(* IEC 61131-3 sources: RL_MAR/experiments/comparison/llm4plc/results/gpt-4o_20260507_114630/20260507_114958, 1 file *)

(* ---- generated_code_iteration_0.st ---- *)
plaintext
START_ST

FUNCTION_BLOCK ShellSortFB
VAR_INPUT
    arr: ARRAY[1..1000] OF DINT; // Input array to be sorted
    sortDirection: BOOL; // Sorting direction (FALSE = ascending, TRUE = descending)
END_VAR

VAR_OUTPUT
    error: BOOL; // Error status (TRUE if an error occurred)
    status: WORD; // Status code
    sorted_arr: ARRAY[1..1000] OF DINT; // Sorted output array
END_VAR

VAR
    state: INT := 0; // Current state of the function block
    N: INT := 1000; // Fixed array size (constant for validation)
    gap: INT; // Gap value for Shell Sort
    i, j: INT; // Loop counters for sorting
    temp: DINT; // Temporary variable for swapping during sorting
END_VAR

// Function block logic
CASE state OF

    // STATE 0: INITIALIZE
    0:
        // Copy input array to output array
        FOR i := 1 TO N DO
            sorted_arr[i] := arr[i];
        END_FOR

        // Validate array size
        IF N <= 1 THEN
            error := TRUE;
            status := 16#8200; // Array size <= 1
            state := 2; // Transition to COMPLETION state
        ELSIF N > 1000 THEN
            error := TRUE;
            status := 16#8201; // Array size > 1000
            state := 2; // Transition to COMPLETION state
        ELSE
            error := FALSE;
            status := 16#0000; // No error
            state := 1; // Transition to SORTING state
        END_IF

    // STATE 1: SORTING
    1:
        // Initialize gap for Shell Sort
        gap := N / 2;

        // Perform Shell Sort
        WHILE gap > 0 DO
            FOR i := gap + 1 TO N DO
                temp := sorted_arr[i];
                j := i;

                // Ascending order sorting
                IF NOT sortDirection THEN
                    WHILE (j > gap) AND (sorted_arr[j - gap] > temp) DO
                        sorted_arr[j] := sorted_arr[j - gap];
                        j := j - gap;
                    END_WHILE;
                // Descending order sorting
                ELSE
                    WHILE (j > gap) AND (sorted_arr[j - gap] < temp) DO
                        sorted_arr[j] := sorted_arr[j - gap];
                        j := j - gap;
                    END_WHILE;
                END_IF;

                sorted_arr[j] := temp;
            END_FOR;

            // Reduce the gap
            gap := gap / 2;
        END_WHILE;

        // Transition to COMPLETION state
        state := 2;

    // STATE 2: COMPLETION
    2:
        // If no error occurred, ensure outputs reflect successful execution
        IF NOT error THEN
            status := 16#0000; // Execution completed without error
        END_IF;

        // Wait for the next execution cycle
        // (No further action required in this state)

END_CASE;

END_FUNCTION_BLOCK

END_ST
